SUBAPPLICATION Automatik_ein (* Subapplication Type *)
  (* Standard: 61499-2 *)
  (* Version 1.0, 2023-02-07, franz *)
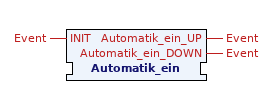
  EVENT_INPUT
    INIT;
  END_EVENT
  EVENT_OUTPUT
    Automatik_ein_UP;
    Automatik_ein_DOWN;
  END_EVENT
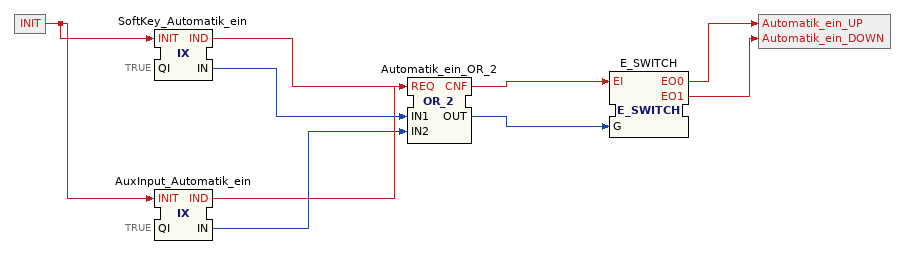
  FBS
    SoftKey_Automatik_ein : IX(QI := TRUE);
    AuxInput_Automatik_ein : IX(QI := TRUE);
    Automatik_ein_OR_2 : OR_2;
    E_SWITCH : E_SWITCH;
  END_FBS
  EVENT_CONNECTIONS
    INIT TO SoftKey_Automatik_ein.INIT;
    INIT TO AuxInput_Automatik_ein.INIT;
    SoftKey_Automatik_ein.IND TO Automatik_ein_OR_2.REQ;
    AuxInput_Automatik_ein.IND TO Automatik_ein_OR_2.REQ;
    Automatik_ein_OR_2.CNF TO E_SWITCH.EI;
    E_SWITCH.EO0 TO Automatik_ein_UP;
    E_SWITCH.EO1 TO Automatik_ein_DOWN;
  END_CONNECTIONS
  DATA_CONNECTIONS
    SoftKey_Automatik_ein.IN TO Automatik_ein_OR_2.IN1;
    AuxInput_Automatik_ein.IN TO Automatik_ein_OR_2.IN2;
    Automatik_ein_OR_2.OUT TO E_SWITCH.G;
  END_CONNECTIONS
END_SUBAPPLICATION
